FUNCTION INTERNAL _SoftCompress
VAR
	i			: UDINT;
	_nFreePtr	: UDINT;
	_stEmpty	: ST_Entry;	
END_VAR

// Find the first free entry in stEntry
FOR i := 1 TO Param.BROADCAST_CAP DO
	IF _Broadcast.stEntry[i].iSignal <> 0 THEN
		i := _Broadcast.stEntry[i].iSignal.id + _Broadcast.stEntry[i].iSignal.size - 1;
	ELSE
		_nFreePtr := i;
	END_IF
END_FOR

// If no free entry found, no need to compress
IF _nFreePtr = 0 THEN
	RETURN;
END_IF 

// Move entries to fill the free space
FOR i := _nFreePtr TO Param.BROADCAST_CAP DO
	IF _Broadcast.stEntry[i].iSignal <> 0 AND_THEN _nFreePtr > 0 THEN
		_Broadcast.stEntry[_nFreePtr] := _Broadcast.stEntry[i];
		_Broadcast.stEntry[i] := _stEmpty;
	ELSE
		_nFreePtr := i;
	END_IF
END_FOR

END_FUNCTION

(* stored: Version 1.1.0.1
   POU _SoftCompress: Id {ca084d12-52fe-4763-b481-46d8da90dfd2}, SpecialFunc None *)
